// ---- VISUs/03_Converters/Conv_handling.TcVIS
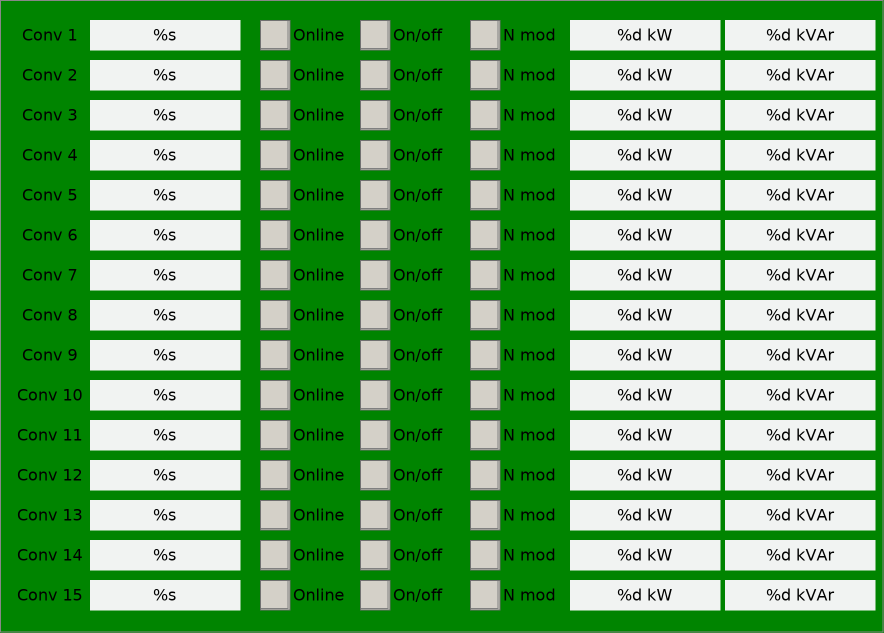
VISUALIZATION Conv_handling  // 884x633
    Rectangle (90,20 150x30), "%s", text variable: GVL_CONV_COMMS.CONVERTERS[1].IP
        OnMouseClick: write the text variable via Default
    Rectangle (10,20 80x30), "Conv 1"
    Rectangle (290,20 60x30), "Online"
    Button (260,20 30x30), colour toggle: GVL_GUI.Conv_online_button[1]
        OnMouseClick: toggle GVL_GUI.Conv_online_button[1]
    Rectangle (390,20 70x30), "On/off"
    Button (360,20 30x30), colour toggle: GVL_GUI.Conv_on_off_button[1]
        OnMouseClick: toggle GVL_GUI.Conv_on_off_button[1]
        OnMouseClick: execute {
            IF GVL_CONV_COMMS.Start_Command[1] = 0 THEN
            	GVL_CONV_COMMS.Comms_Control_Word[1]:= GVL_CONV_COMMS.Comms_Control_Word[1] OR 16#0001;
            ELSE
            	GVL_CONV_COMMS.Comms_Control_Word[1]:= GVL_CONV_COMMS.Comms_Control_Word[1] AND 16#FFFE;
            END_IF
        }
    Rectangle (500,20 70x30), "N mod"
    Button (470,20 30x30), colour toggle: GVL_GUI.Conv_n_mode_button[1]
        OnMouseClick: toggle GVL_GUI.Conv_n_mode_button[1]
        OnMouseClick: execute {
            IF GVL_CONV_COMMS.Night_Mode_Active[1] = 0 THEN
            	GVL_CONV_COMMS.Comms_Control_Word[1]:= GVL_CONV_COMMS.Comms_Control_Word[1] OR 16#0002;
            ELSE
            	GVL_CONV_COMMS.Comms_Control_Word[1]:= GVL_CONV_COMMS.Comms_Control_Word[1] AND 16#FFFD;
            END_IF
        }
    Rectangle (90,60 150x30), "%s", text variable: GVL_CONV_COMMS.CONVERTERS[2].IP
        OnMouseClick: write the text variable via Default
    Rectangle (10,60 80x30), "Conv 2"
    Rectangle (290,60 60x30), "Online"
    Button (260,60 30x30), colour toggle: GVL_GUI.Conv_online_button[2]
        OnMouseClick: toggle GVL_GUI.Conv_online_button[2]
    Rectangle (390,60 70x30), "On/off"
    Button (360,60 30x30), colour toggle: GVL_GUI.Conv_on_off_button[2]
        OnMouseClick: toggle GVL_GUI.Conv_on_off_button[2]
        OnMouseClick: execute {
            IF GVL_CONV_COMMS.Start_Command[2] = 0 THEN
            	GVL_CONV_COMMS.Comms_Control_Word[2]:= GVL_CONV_COMMS.Comms_Control_Word[2] or 16#0001;
            ELSE
            	GVL_CONV_COMMS.Comms_Control_Word[2]:= GVL_CONV_COMMS.Comms_Control_Word[2] AND 16#FFFE;
            END_IF
        }
    Rectangle (500,60 70x30), "N mod"
    Button (470,60 30x30), colour toggle: GVL_GUI.Conv_n_mode_button[2]
        OnMouseClick: toggle GVL_GUI.Conv_n_mode_button[2]
        OnMouseClick: execute {
            IF GVL_CONV_COMMS.Night_Mode_Active[2] = 0 THEN
            	GVL_CONV_COMMS.Comms_Control_Word[2]:= GVL_CONV_COMMS.Comms_Control_Word[2] or 16#0002;
            ELSE
            	GVL_CONV_COMMS.Comms_Control_Word[2]:= GVL_CONV_COMMS.Comms_Control_Word[2] AND 16#FFFD;
            END_IF
        }
    Rectangle (90,100 150x30), "%s", text variable: GVL_CONV_COMMS.CONVERTERS[3].IP
        OnMouseClick: write the text variable via Default
    Rectangle (10,100 80x30), "Conv 3"
    Rectangle (290,100 60x30), "Online"
    Button (260,100 30x30), colour toggle: GVL_GUI.Conv_online_button[3]
        OnMouseClick: toggle GVL_GUI.Conv_online_button[3]
    Rectangle (390,100 70x30), "On/off"
    Button (360,100 30x30), colour toggle: GVL_GUI.Conv_on_off_button[3]
        OnMouseClick: toggle GVL_GUI.Conv_on_off_button[3]
        OnMouseClick: execute {
            IF GVL_CONV_COMMS.Start_Command[3] = 0 THEN
            	GVL_CONV_COMMS.Comms_Control_Word[3]:= GVL_CONV_COMMS.Comms_Control_Word[3] or 16#0001;
            ELSE
            	GVL_CONV_COMMS.Comms_Control_Word[3]:= GVL_CONV_COMMS.Comms_Control_Word[3] AND 16#FFFE;
            END_IF
        }
    Rectangle (500,100 70x30), "N mod"
    Button (470,100 30x30), colour toggle: GVL_GUI.Conv_n_mode_button[3]
        OnMouseClick: toggle GVL_GUI.Conv_n_mode_button[3]
        OnMouseClick: execute {
            IF GVL_CONV_COMMS.Night_Mode_Active[3] = 0 THEN
            	GVL_CONV_COMMS.Comms_Control_Word[3]:= GVL_CONV_COMMS.Comms_Control_Word[3] OR 16#0002;
            ELSE
            	GVL_CONV_COMMS.Comms_Control_Word[3]:= GVL_CONV_COMMS.Comms_Control_Word[3] AND 16#FFFD;
            END_IF
        }
    Rectangle (90,140 150x30), "%s", text variable: GVL_CONV_COMMS.CONVERTERS[4].IP
        OnMouseClick: write the text variable via Default
    Rectangle (10,140 80x30), "Conv 4"
    Rectangle (290,140 60x30), "Online"
    Button (260,140 30x30), colour toggle: GVL_GUI.Conv_online_button[4]
        OnMouseClick: toggle GVL_GUI.Conv_online_button[4]
    Rectangle (390,140 70x30), "On/off"
    Button (360,140 30x30), colour toggle: GVL_GUI.Conv_on_off_button[4]
        OnMouseClick: toggle GVL_GUI.Conv_on_off_button[4]
        OnMouseClick: execute {
            IF GVL_CONV_COMMS.Start_Command[4] = 0 THEN
            	GVL_CONV_COMMS.Comms_Control_Word[4]:= GVL_CONV_COMMS.Comms_Control_Word[4] OR 16#0001;
            ELSE
            	GVL_CONV_COMMS.Comms_Control_Word[4]:= GVL_CONV_COMMS.Comms_Control_Word[4] AND 16#FFFE;
            END_IF
        }
    Rectangle (500,140 70x30), "N mod"
    Button (470,140 30x30), colour toggle: GVL_GUI.Conv_n_mode_button[4]
        OnMouseClick: toggle GVL_GUI.Conv_n_mode_button[4]
        OnMouseClick: execute {
            IF GVL_CONV_COMMS.Night_Mode_Active[4] = 0 THEN
            	GVL_CONV_COMMS.Comms_Control_Word[4]:= GVL_CONV_COMMS.Comms_Control_Word[4] OR 16#0002;
            ELSE
            	GVL_CONV_COMMS.Comms_Control_Word[4]:= GVL_CONV_COMMS.Comms_Control_Word[4] AND 16#FFFD;
            END_IF
        }
    Rectangle (90,180 150x30), "%s", text variable: GVL_CONV_COMMS.CONVERTERS[5].IP
        OnMouseClick: write the text variable via Default
    Rectangle (10,180 80x30), "Conv 5"
    Rectangle (290,180 60x30), "Online"
    Button (260,180 30x30), colour toggle: GVL_GUI.Conv_online_button[5]
        OnMouseClick: toggle GVL_GUI.Conv_online_button[5]
    Rectangle (390,180 70x30), "On/off"
    Button (360,180 30x30), colour toggle: GVL_GUI.Conv_on_off_button[5]
        OnMouseClick: toggle GVL_GUI.Conv_on_off_button[5]
        OnMouseClick: execute {
            IF GVL_CONV_COMMS.Start_Command[5] = 0 THEN
            	GVL_CONV_COMMS.Comms_Control_Word[5]:= GVL_CONV_COMMS.Comms_Control_Word[5] OR 16#0001;
            ELSE
            	GVL_CONV_COMMS.Comms_Control_Word[5]:= GVL_CONV_COMMS.Comms_Control_Word[5] AND 16#FFFE;
            END_IF
        }
    Rectangle (500,180 70x30), "N mod"
    Button (470,180 30x30), colour toggle: GVL_GUI.Conv_n_mode_button[5]
        OnMouseClick: toggle GVL_GUI.Conv_n_mode_button[5]
        OnMouseClick: execute {
            IF GVL_CONV_COMMS.Night_Mode_Active[5] = 0 THEN
            	GVL_CONV_COMMS.Comms_Control_Word[5]:= GVL_CONV_COMMS.Comms_Control_Word[5] OR 16#0002;
            ELSE
            	GVL_CONV_COMMS.Comms_Control_Word[5]:= GVL_CONV_COMMS.Comms_Control_Word[5] AND 16#FFFD;
            END_IF
        }
    Rectangle (90,220 150x30), "%s", text variable: GVL_CONV_COMMS.CONVERTERS[6].IP
        OnMouseClick: write the text variable via Default
    Rectangle (10,220 80x30), "Conv 6"
    Rectangle (290,220 60x30), "Online"
    Button (260,220 30x30), colour toggle: GVL_GUI.Conv_online_button[6]
        OnMouseClick: toggle GVL_GUI.Conv_online_button[6]
    Rectangle (390,220 70x30), "On/off"
    Button (360,220 30x30), colour toggle: GVL_GUI.Conv_on_off_button[6]
        OnMouseClick: toggle GVL_GUI.Conv_on_off_button[6]
        OnMouseClick: execute {
            IF GVL_CONV_COMMS.Start_Command[6] = 0 THEN
            	GVL_CONV_COMMS.Comms_Control_Word[6]:= GVL_CONV_COMMS.Comms_Control_Word[6] OR 16#0001;
            ELSE
            	GVL_CONV_COMMS.Comms_Control_Word[6]:= GVL_CONV_COMMS.Comms_Control_Word[6] AND 16#FFFE;
            END_IF
        }
    Rectangle (500,220 70x30), "N mod"
    Button (470,220 30x30), colour toggle: GVL_GUI.Conv_n_mode_button[6]
        OnMouseClick: toggle GVL_GUI.Conv_n_mode_button[6]
        OnMouseClick: execute {
            IF GVL_CONV_COMMS.Night_Mode_Active[6] = 0 THEN
            	GVL_CONV_COMMS.Comms_Control_Word[6]:= GVL_CONV_COMMS.Comms_Control_Word[6] OR 16#0002;
            ELSE
            	GVL_CONV_COMMS.Comms_Control_Word[6]:= GVL_CONV_COMMS.Comms_Control_Word[6] AND 16#FFFD;
            END_IF
        }
    Rectangle (90,260 150x30), "%s", text variable: GVL_CONV_COMMS.CONVERTERS[7].IP
        OnMouseClick: write the text variable via Default
    Rectangle (10,260 80x30), "Conv 7"
    Rectangle (290,260 60x30), "Online"
    Button (260,260 30x30), colour toggle: GVL_GUI.Conv_online_button[7]
        OnMouseClick: toggle GVL_GUI.Conv_online_button[7]
    Rectangle (390,260 70x30), "On/off"
    Button (360,260 30x30), colour toggle: GVL_GUI.Conv_on_off_button[7]
        OnMouseClick: toggle GVL_GUI.Conv_on_off_button[7]
        OnMouseClick: execute {
            IF GVL_CONV_COMMS.Start_Command[7] = 0 THEN
            	GVL_CONV_COMMS.Comms_Control_Word[7]:= GVL_CONV_COMMS.Comms_Control_Word[7] OR 16#0001;
            ELSE
            	GVL_CONV_COMMS.Comms_Control_Word[7]:= GVL_CONV_COMMS.Comms_Control_Word[7] AND 16#FFFE;
            END_IF
        }
    Rectangle (500,260 70x30), "N mod"
    Button (470,260 30x30), colour toggle: GVL_GUI.Conv_n_mode_button[7]
        OnMouseClick: toggle GVL_GUI.Conv_n_mode_button[7]
        OnMouseClick: execute {
            IF GVL_CONV_COMMS.Night_Mode_Active[7] = 0 THEN
            	GVL_CONV_COMMS.Comms_Control_Word[7]:= GVL_CONV_COMMS.Comms_Control_Word[7] OR 16#0002;
            ELSE
            	GVL_CONV_COMMS.Comms_Control_Word[7]:= GVL_CONV_COMMS.Comms_Control_Word[7] AND 16#FFFD;
            END_IF
        }
    Rectangle (90,300 150x30), "%s", text variable: GVL_CONV_COMMS.CONVERTERS[8].IP
        OnMouseClick: write the text variable via Default
    Rectangle (10,300 80x30), "Conv 8"
    Rectangle (290,300 60x30), "Online"
    Button (260,300 30x30), colour toggle: GVL_GUI.Conv_online_button[8]
        OnMouseClick: toggle GVL_GUI.Conv_online_button[8]
    Rectangle (390,300 70x30), "On/off"
    Button (360,300 30x30), colour toggle: GVL_GUI.Conv_on_off_button[8]
        OnMouseClick: toggle GVL_GUI.Conv_on_off_button[8]
        OnMouseClick: execute {
            IF GVL_CONV_COMMS.Start_Command[8] = 0 THEN
            	GVL_CONV_COMMS.Comms_Control_Word[8]:= GVL_CONV_COMMS.Comms_Control_Word[8] OR 16#0001;
            ELSE
            	GVL_CONV_COMMS.Comms_Control_Word[8]:= GVL_CONV_COMMS.Comms_Control_Word[8] AND 16#FFFE;
            END_IF
        }
    Rectangle (500,300 70x30), "N mod"
    Button (470,300 30x30), colour toggle: GVL_GUI.Conv_n_mode_button[8]
        OnMouseClick: toggle GVL_GUI.Conv_n_mode_button[8]
        OnMouseClick: execute {
            IF GVL_CONV_COMMS.Night_Mode_Active[8] = 0 THEN
            	GVL_CONV_COMMS.Comms_Control_Word[8]:= GVL_CONV_COMMS.Comms_Control_Word[8] OR 16#0002;
            ELSE
            	GVL_CONV_COMMS.Comms_Control_Word[8]:= GVL_CONV_COMMS.Comms_Control_Word[8] AND 16#FFFD;
            END_IF
        }
    Rectangle (90,340 150x30), "%s", text variable: GVL_CONV_COMMS.CONVERTERS[9].IP
        OnMouseClick: write the text variable via Default
    Rectangle (10,340 80x30), "Conv 9"
    Rectangle (290,340 60x30), "Online"
    Button (260,340 30x30), colour toggle: GVL_GUI.Conv_online_button[9]
        OnMouseClick: toggle GVL_GUI.Conv_online_button[9]
    Rectangle (390,340 70x30), "On/off"
    Button (360,340 30x30), colour toggle: GVL_GUI.Conv_on_off_button[9]
        OnMouseClick: toggle GVL_GUI.Conv_on_off_button[9]
        OnMouseClick: execute {
            IF GVL_CONV_COMMS.Start_Command[9] = 0 THEN
            	GVL_CONV_COMMS.Comms_Control_Word[9]:= GVL_CONV_COMMS.Comms_Control_Word[9] OR 16#0001;
            ELSE
            	GVL_CONV_COMMS.Comms_Control_Word[9]:= GVL_CONV_COMMS.Comms_Control_Word[9] AND 16#FFFE;
            END_IF
        }
    Rectangle (500,340 70x30), "N mod"
    Button (470,340 30x30), colour toggle: GVL_GUI.Conv_n_mode_button[9]
        OnMouseClick: toggle GVL_GUI.Conv_n_mode_button[9]
        OnMouseClick: execute {
            IF GVL_CONV_COMMS.Night_Mode_Active[9] = 0 THEN
            	GVL_CONV_COMMS.Comms_Control_Word[9]:= GVL_CONV_COMMS.Comms_Control_Word[9] OR 16#0002;
            ELSE
            	GVL_CONV_COMMS.Comms_Control_Word[9]:= GVL_CONV_COMMS.Comms_Control_Word[9] AND 16#FFFD;
            END_IF
        }
    Rectangle (90,380 150x30), "%s", text variable: GVL_CONV_COMMS.CONVERTERS[10].IP
        OnMouseClick: write the text variable via Default
    Rectangle (10,380 80x30), "Conv 10"
    Rectangle (290,380 60x30), "Online"
    Button (260,380 30x30), colour toggle: GVL_GUI.Conv_online_button[10]
        OnMouseClick: toggle GVL_GUI.Conv_online_button[10]
    Rectangle (390,380 70x30), "On/off"
    Button (360,380 30x30), colour toggle: GVL_GUI.Conv_on_off_button[10]
        OnMouseClick: toggle GVL_GUI.Conv_on_off_button[10]
        OnMouseClick: execute {
            IF GVL_CONV_COMMS.Start_Command[10] = 0 THEN
            	GVL_CONV_COMMS.Comms_Control_Word[10]:= GVL_CONV_COMMS.Comms_Control_Word[10] OR 16#0001;
            ELSE
            	GVL_CONV_COMMS.Comms_Control_Word[10]:= GVL_CONV_COMMS.Comms_Control_Word[10] AND 16#FFFE;
            END_IF
        }
    Rectangle (500,380 70x30), "N mod"
    Button (470,380 30x30), colour toggle: GVL_GUI.Conv_n_mode_button[10]
        OnMouseClick: toggle GVL_GUI.Conv_n_mode_button[10]
        OnMouseClick: execute {
            IF GVL_CONV_COMMS.Night_Mode_Active[10] = 0 THEN
            	GVL_CONV_COMMS.Comms_Control_Word[10]:= GVL_CONV_COMMS.Comms_Control_Word[10] OR 16#0002;
            ELSE
            	GVL_CONV_COMMS.Comms_Control_Word[10]:= GVL_CONV_COMMS.Comms_Control_Word[10] AND 16#FFFD;
            END_IF
        }
    Rectangle (90,420 150x30), "%s", text variable: GVL_CONV_COMMS.CONVERTERS[11].IP
        OnMouseClick: write the text variable via Default
    Rectangle (10,420 80x30), "Conv 11"
    Rectangle (290,420 60x30), "Online"
    Button (260,420 30x30), colour toggle: GVL_GUI.Conv_online_button[11]
        OnMouseClick: toggle GVL_GUI.Conv_online_button[11]
    Rectangle (390,420 70x30), "On/off"
    Button (360,420 30x30), colour toggle: GVL_GUI.Conv_on_off_button[11]
        OnMouseClick: toggle GVL_GUI.Conv_on_off_button[11]
        OnMouseClick: execute {
            IF GVL_CONV_COMMS.Start_Command[11] = 0 THEN
            	GVL_CONV_COMMS.Comms_Control_Word[11]:= GVL_CONV_COMMS.Comms_Control_Word[11] OR 16#0001;
            ELSE
            	GVL_CONV_COMMS.Comms_Control_Word[11]:= GVL_CONV_COMMS.Comms_Control_Word[11] AND 16#FFFE;
            END_IF
        }
    Rectangle (500,420 70x30), "N mod"
    Button (470,420 30x30), colour toggle: GVL_GUI.Conv_n_mode_button[11]
        OnMouseClick: toggle GVL_GUI.Conv_n_mode_button[11]
        OnMouseClick: execute {
            IF GVL_CONV_COMMS.Night_Mode_Active[11] = 0 THEN
            	GVL_CONV_COMMS.Comms_Control_Word[11]:= GVL_CONV_COMMS.Comms_Control_Word[11] OR 16#0002;
            ELSE
            	GVL_CONV_COMMS.Comms_Control_Word[11]:= GVL_CONV_COMMS.Comms_Control_Word[11] AND 16#FFFD;
            END_IF
        }
    Rectangle (90,460 150x30), "%s", text variable: GVL_CONV_COMMS.CONVERTERS[12].IP
        OnMouseClick: write the text variable via Default
    Rectangle (10,460 80x30), "Conv 12"
    Rectangle (290,460 60x30), "Online"
    Button (260,460 30x30), colour toggle: GVL_GUI.Conv_online_button[12]
        OnMouseClick: toggle GVL_GUI.Conv_online_button[12]
    Rectangle (390,460 70x30), "On/off"
    Button (360,460 30x30), colour toggle: GVL_GUI.Conv_on_off_button[12]
        OnMouseClick: toggle GVL_GUI.Conv_on_off_button[12]
        OnMouseClick: execute {
            IF GVL_CONV_COMMS.Start_Command[12] = 0 THEN
            	GVL_CONV_COMMS.Comms_Control_Word[12]:= GVL_CONV_COMMS.Comms_Control_Word[12] OR 16#0001;
            ELSE
            	GVL_CONV_COMMS.Comms_Control_Word[12]:= GVL_CONV_COMMS.Comms_Control_Word[12] AND 16#FFFE;
            END_IF
        }
    Rectangle (500,460 70x30), "N mod"
    Button (470,460 30x30), colour toggle: GVL_GUI.Conv_n_mode_button[12]
        OnMouseClick: toggle GVL_GUI.Conv_n_mode_button[12]
        OnMouseClick: execute {
            IF GVL_CONV_COMMS.Night_Mode_Active[12] = 0 THEN
            	GVL_CONV_COMMS.Comms_Control_Word[12]:= GVL_CONV_COMMS.Comms_Control_Word[12] OR 16#0002;
            ELSE
            	GVL_CONV_COMMS.Comms_Control_Word[12]:= GVL_CONV_COMMS.Comms_Control_Word[12] AND 16#FFFD;
            END_IF
        }
    Rectangle (90,500 150x30), "%s", text variable: GVL_CONV_COMMS.CONVERTERS[13].IP
        OnMouseClick: write the text variable via Default
    Rectangle (10,500 80x30), "Conv 13"
    Rectangle (290,500 60x30), "Online"
    Button (260,500 30x30), colour toggle: GVL_GUI.Conv_online_button[13]
        OnMouseClick: toggle GVL_GUI.Conv_online_button[13]
    Rectangle (390,500 70x30), "On/off"
    Button (360,500 30x30), colour toggle: GVL_GUI.Conv_on_off_button[13]
        OnMouseClick: toggle GVL_GUI.Conv_on_off_button[13]
        OnMouseClick: execute {
            IF GVL_CONV_COMMS.Start_Command[13] = 0 THEN
            	GVL_CONV_COMMS.Comms_Control_Word[13]:= GVL_CONV_COMMS.Comms_Control_Word[13] OR 16#0001;
            ELSE
            	GVL_CONV_COMMS.Comms_Control_Word[13]:= GVL_CONV_COMMS.Comms_Control_Word[13] AND 16#FFFE;
            END_IF
        }
    Rectangle (500,500 70x30), "N mod"
    Button (470,500 30x30), colour toggle: GVL_GUI.Conv_n_mode_button[13]
        OnMouseClick: toggle GVL_GUI.Conv_n_mode_button[13]
        OnMouseClick: execute {
            IF GVL_CONV_COMMS.Night_Mode_Active[13] = 0 THEN
            	GVL_CONV_COMMS.Comms_Control_Word[13]:= GVL_CONV_COMMS.Comms_Control_Word[13] OR 16#0002;
            ELSE
            	GVL_CONV_COMMS.Comms_Control_Word[13]:= GVL_CONV_COMMS.Comms_Control_Word[13] AND 16#FFFD;
            END_IF
        }
    Rectangle (90,540 150x30), "%s", text variable: GVL_CONV_COMMS.CONVERTERS[14].IP
        OnMouseClick: write the text variable via Default
    Rectangle (10,540 80x30), "Conv 14"
    Rectangle (290,540 60x30), "Online"
    Button (260,540 30x30), colour toggle: GVL_GUI.Conv_online_button[14]
        OnMouseClick: toggle GVL_GUI.Conv_online_button[14]
    Rectangle (390,540 70x30), "On/off"
    Button (360,540 30x30), colour toggle: GVL_GUI.Conv_on_off_button[14]
        OnMouseClick: toggle GVL_GUI.Conv_on_off_button[14]
        OnMouseClick: execute {
            IF GVL_CONV_COMMS.Start_Command[14] = 0 THEN
            	GVL_CONV_COMMS.Comms_Control_Word[14]:= GVL_CONV_COMMS.Comms_Control_Word[14] OR 16#0001;
            ELSE
            	GVL_CONV_COMMS.Comms_Control_Word[14]:= GVL_CONV_COMMS.Comms_Control_Word[14] AND 16#FFFE;
            END_IF
        }
    Rectangle (500,540 70x30), "N mod"
    Button (470,540 30x30), colour toggle: GVL_GUI.Conv_n_mode_button[14]
        OnMouseClick: toggle GVL_GUI.Conv_n_mode_button[14]
        OnMouseClick: execute {
            IF GVL_CONV_COMMS.Night_Mode_Active[14] = 0 THEN
            	GVL_CONV_COMMS.Comms_Control_Word[14]:= GVL_CONV_COMMS.Comms_Control_Word[14] OR 16#0002;
            ELSE
            	GVL_CONV_COMMS.Comms_Control_Word[14]:= GVL_CONV_COMMS.Comms_Control_Word[14] AND 16#FFFD;
            END_IF
        }
    Rectangle (90,580 150x30), "%s", text variable: GVL_CONV_COMMS.CONVERTERS[15].IP
        OnMouseClick: write the text variable via Default
    Rectangle (10,580 80x30), "Conv 15"
    Rectangle (290,580 60x30), "Online"
    Button (260,580 30x30), colour toggle: GVL_GUI.Conv_online_button[15]
        OnMouseClick: toggle GVL_GUI.Conv_online_button[15]
    Rectangle (390,580 70x30), "On/off"
    Button (360,580 30x30), colour toggle: GVL_GUI.Conv_on_off_button[15]
        OnMouseClick: toggle GVL_GUI.Conv_on_off_button[15]
        OnMouseClick: execute {
            IF GVL_CONV_COMMS.Start_Command[15] = 0 THEN
            	GVL_CONV_COMMS.Comms_Control_Word[15]:= GVL_CONV_COMMS.Comms_Control_Word[15] OR 16#0001;
            ELSE
            	GVL_CONV_COMMS.Comms_Control_Word[15]:= GVL_CONV_COMMS.Comms_Control_Word[15] AND 16#FFFE;
            END_IF
        }
    Rectangle (500,580 70x30), "N mod"
    Button (470,580 30x30), colour toggle: GVL_GUI.Conv_n_mode_button[15]
        OnMouseClick: toggle GVL_GUI.Conv_n_mode_button[15]
        OnMouseClick: execute {
            IF GVL_CONV_COMMS.Night_Mode_Active[15] = 0 THEN
            	GVL_CONV_COMMS.Comms_Control_Word[15]:= GVL_CONV_COMMS.Comms_Control_Word[15] OR 16#0002;
            ELSE
            	GVL_CONV_COMMS.Comms_Control_Word[15]:= GVL_CONV_COMMS.Comms_Control_Word[15] AND 16#FFFD;
            END_IF
        }
    Rectangle (570,20 150x30), "%d kW", text variable: GVL_CONV_COMMS.P_Measured[1]
    Rectangle (725,20 150x30), "%d kVAr", text variable: GVL_CONV_COMMS.Q_Measured[1]
    Rectangle (570,60 150x30), "%d kW", text variable: GVL_CONV_COMMS.P_Measured[2]
    Rectangle (725,60 150x30), "%d kVAr", text variable: GVL_CONV_COMMS.Q_Measured[2]
    Rectangle (570,100 150x30), "%d kW", text variable: GVL_CONV_COMMS.P_Measured[3]
    Rectangle (725,100 150x30), "%d kVAr", text variable: GVL_CONV_COMMS.Q_Measured[3]
    Rectangle (570,140 150x30), "%d kW", text variable: GVL_CONV_COMMS.P_Measured[4]
    Rectangle (725,140 150x30), "%d kVAr", text variable: GVL_CONV_COMMS.Q_Measured[4]
    Rectangle (570,180 150x30), "%d kW", text variable: GVL_CONV_COMMS.P_Measured[5]
    Rectangle (725,180 150x30), "%d kVAr", text variable: GVL_CONV_COMMS.Q_Measured[5]
    Rectangle (570,220 150x30), "%d kW", text variable: GVL_CONV_COMMS.P_Measured[6]
    Rectangle (725,220 150x30), "%d kVAr", text variable: GVL_CONV_COMMS.Q_Measured[6]
    Rectangle (570,260 150x30), "%d kW", text variable: GVL_CONV_COMMS.P_Measured[7]
    Rectangle (725,260 150x30), "%d kVAr", text variable: GVL_CONV_COMMS.Q_Measured[7]
    Rectangle (570,300 150x30), "%d kW", text variable: GVL_CONV_COMMS.P_Measured[8]
    Rectangle (725,300 150x30), "%d kVAr", text variable: GVL_CONV_COMMS.Q_Measured[8]
    Rectangle (570,340 150x30), "%d kW", text variable: GVL_CONV_COMMS.P_Measured[9]
    Rectangle (725,340 150x30), "%d kVAr", text variable: GVL_CONV_COMMS.Q_Measured[9]
    Rectangle (570,380 150x30), "%d kW", text variable: GVL_CONV_COMMS.P_Measured[10]
    Rectangle (725,380 150x30), "%d kVAr", text variable: GVL_CONV_COMMS.Q_Measured[10]
    Rectangle (570,420 150x30), "%d kW", text variable: GVL_CONV_COMMS.P_Measured[11]
    Rectangle (725,420 150x30), "%d kVAr", text variable: GVL_CONV_COMMS.Q_Measured[11]
    Rectangle (570,460 150x30), "%d kW", text variable: GVL_CONV_COMMS.P_Measured[12]
    Rectangle (725,460 150x30), "%d kVAr", text variable: GVL_CONV_COMMS.Q_Measured[12]
    Rectangle (570,500 150x30), "%d kW", text variable: GVL_CONV_COMMS.P_Measured[13]
    Rectangle (725,500 150x30), "%d kVAr", text variable: GVL_CONV_COMMS.Q_Measured[13]
    Rectangle (570,540 150x30), "%d kW", text variable: GVL_CONV_COMMS.P_Measured[14]
    Rectangle (725,540 150x30), "%d kVAr", text variable: GVL_CONV_COMMS.Q_Measured[14]
    Rectangle (570,580 150x30), "%d kW", text variable: GVL_CONV_COMMS.P_Measured[15]
    Rectangle (725,580 150x30), "%d kVAr", text variable: GVL_CONV_COMMS.Q_Measured[5]
END_VISUALIZATION

// ---- VISUs/04_Powermeter/M_board_status.TcTLO
TEXTLIST M_board_status
  0 = 'Offline'
  1 = 'Online'
   = ''
END_TEXTLIST

// ---- VISUs/04_Powermeter/PM_config.TcVIS
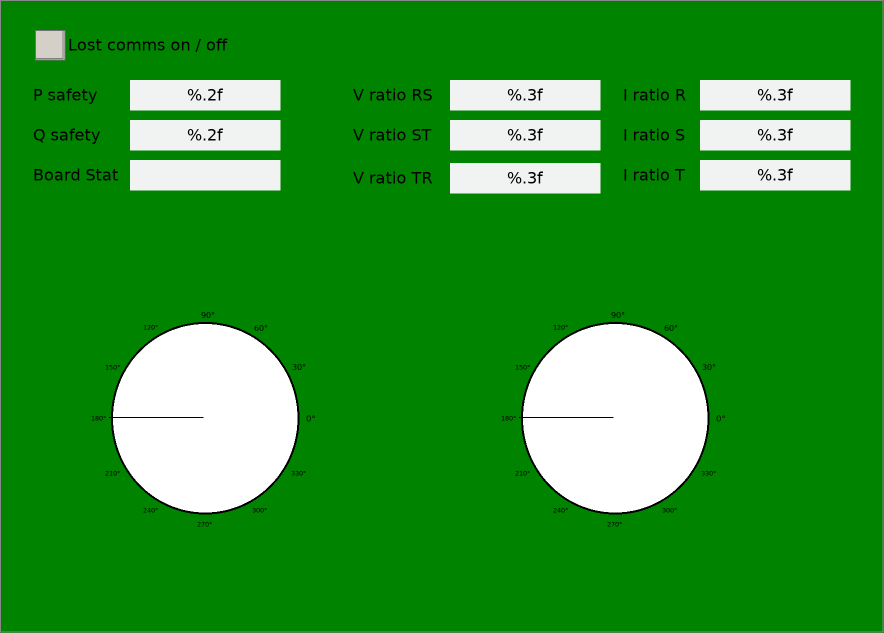
VISUALIZATION PM_config  // 884x633
    Rectangle (350,80 92x30), "V ratio RS"
    Rectangle (450,80 150x30), "%.3f", text variable: GVL_HANDLER.GUI_vars[V_ratio_RS]
        OnMouseClick: write the text variable via Default
    Rectangle (350,120 92x30), "V ratio ST"
    Rectangle (450,120 150x30), "%.3f", text variable: GVL_HANDLER.GUI_vars[V_ratio_ST]
        OnMouseClick: write the text variable via Default
    Rectangle (350,163 92x30), "V ratio TR"
    Rectangle (450,163 150x30), "%.3f", text variable: GVL_HANDLER.GUI_vars[V_ratio_TR]
        OnMouseClick: write the text variable via Default
    Rectangle (620,80 92x30), "I ratio R"
    Rectangle (700,80 150x30), "%.3f", text variable: GVL_HANDLER.GUI_vars[I_ratio_R]
        OnMouseClick: write the text variable via Default
    Rectangle (620,120 92x30), "I ratio S"
    Rectangle (700,120 150x30), "%.3f", text variable: GVL_HANDLER.GUI_vars[I_ratio_S]
        OnMouseClick: write the text variable via Default
    Rectangle (620,160 92x30), "I ratio T"
    Rectangle (700,160 150x30), "%.3f", text variable: GVL_HANDLER.GUI_vars[I_ratio_T]
        OnMouseClick: write the text variable via Default
    Ellipse (111,322 188x192)
    Line (109,417) (203,417)
        p2858320360: GVL_POWERMETER.M_board_I_L1_angle
        p1097714728: GVL_POWERMETER.I_L1_pu
    Line (109,417) (203,417)
        p2858320360: GVL_POWERMETER.M_board_I_L3_angle
        p1097714728: GVL_POWERMETER.I_L3_pu
    Line (109,417) (203,417)
        p2858320360: GVL_POWERMETER.M_board_I_L2_angle
        p1097714728: GVL_POWERMETER.I_L2_pu
    Textfield (291,362 16x11), "30°"
    Textfield (253,323 16x11), "60°"
    Textfield (200,310 16x11), "90°"
    Textfield (142,322 18x11), "120°"
    Textfield (104,362 18x11), "150°"
    Textfield (90,413 18x11), "180°"
    Textfield (302,413 18x11), "0°"
    Textfield (104,468 18x11), "210°"
    Textfield (142,505 18x11), "240°"
    Textfield (196,519 18x11), "270°"
    Textfield (251,505 18x11), "300°"
    Textfield (290,468 18x11), "330°"
    Ellipse (521,322 188x192)
    Line (519,417) (613,417)
        p1097714728: GVL_POWERMETER.V_L1N_pu
    Line (519,417) (613,417)
        p2858320360: -GVL_POWERMETER.Power_analyzer.V_L1L3_angle
        p1097714728: GVL_POWERMETER.V_L3N_pu
    Line (519,417) (613,417)
        p2858320360: GVL_POWERMETER.Power_analyzer.V_L1L2_angle
        p1097714728: GVL_POWERMETER.V_L2N_pu
    Textfield (701,362 16x11), "30°"
    Textfield (663,323 16x11), "60°"
    Textfield (610,310 16x11), "90°"
    Textfield (552,322 18x11), "120°"
    Textfield (514,362 18x11), "150°"
    Textfield (500,413 18x11), "180°"
    Textfield (712,413 18x11), "0°"
    Textfield (514,468 18x11), "210°"
    Textfield (552,505 18x11), "240°"
    Textfield (606,519 18x11), "270°"
    Textfield (661,505 18x11), "300°"
    Textfield (700,468 18x11), "330°"
    Rectangle (65,30 160x30), "Lost comms on / off"
    Button (35,30 30x30), colour toggle: GVL_POWERMETER.Alg_lost_comms_enable
        OnMouseClick: toggle GVL_HANDLER.GUI_vars[Lost_comms_enable]
    Rectangle (130,80 150x30), "%.2f", text variable: GVL_HANDLER.GUI_vars[P_safety]
        OnMouseClick: write the text variable via Default
    Rectangle (30,80 92x30), "P safety"
    Rectangle (130,120 150x30), "%.2f", text variable: GVL_HANDLER.GUI_vars[Q_safety]
        OnMouseClick: write the text variable via Default
    Rectangle (30,120 92x30), "Q safety"
    Rectangle (130,160 150x30), text list: 'M_board_status'
    Rectangle (30,160 100x30), "Board Stat"
END_VISUALIZATION
